{attribute 'GeneratedUsingTerminal: EL1259-0000-0016'}
{attribute addProperty BoxType "EL1259-0000-0016"}
{attribute addProperty Id "Output_buffer_resetBOOL1Manual_output_stateBOOL1Force_orderBOOL1Output_order_counterUSINT1No_of_output_eventsUSINT1"}
{attribute addProperty CRC "2959048927"}
{attribute addProperty Size "5"}
TYPE Ctrl_B05F80DF :
STRUCT
	{attribute addProperty Name "Output_buffer_reset"}
	Output_buffer_reset : BOOL;
	{attribute addProperty Name "Manual_output_state"}
	Manual_output_state : BOOL;
	{attribute addProperty Name "Force_order"}
	Force_order : BOOL;
	{attribute addProperty Name "Output_order_counter"}
	Output_order_counter : USINT;
	{attribute addProperty Name "No_of_output_events"}
	No_of_output_events : USINT;
END_STRUCT
END_TYPE

(* stored: Version 1.2.0.0, ProductVersion 3.1.4024.9
   DUT Ctrl_B05F80DF: Id {4b6d3f8d-03f2-48af-8e4b-4302a575e9df} *)
